{attribute 'linkalways'} 
{attribute 'no_explicit_call' := 'This FB is a CLASS and must be accessed using methods or properties'}
{attribute 'enable_dynamic_creation'}
FUNCTION_BLOCK PUBLIC DummyCommand EXTENDS AsyncCommand
VAR
	id : DINT;
	name : T_MaxString;
	timer : Ton;
END_VAR

METHOD PRIVATE AdsLog
VAR_INPUT
	message : T_MaxString;
END_VAR
VAR
	arrghhhh : T_MaxString := '%s';
END_VAR
VAR_INST
	format : FB_FormatString;
END_VAR
format(
	sFormat := 'DummyCommand{id=%d, name=%s} -> %s',
	arg1 := F_DInt(id),
	arg2 := F_String(name),
	arg3 := F_String(arrghhhh)
);

AdsLogStr(
	msgCtrlMask := ADSLOG_MSGTYPE_HINT,
	msgFmtStr := format.sOut,
	strArg := message
);
END_METHOD

METHOD FB_init : BOOL
VAR_INPUT
	bInitRetains : BOOL; // if TRUE, the retain variables are initialized (warm start / cold start)
	bInCopyCode : BOOL;  // if TRUE, the instance afterwards gets moved into the copy code (online change)
	id : DINT;
	name : T_MaxString;
END_VAR
THIS^.id := id;
THIS^.name := name;

AdsLog('FB_init');
END_METHOD

METHOD PROTECTED OnAborted
AdsLog('Aborted');
END_METHOD

METHOD PROTECTED OnAborting
VAR_INPUT
	stateControl : I_AsyncCommandStateControl;
END_VAR
AdsLog('Aborting');

WrapItUp(stateControl);
END_METHOD

METHOD PROTECTED OnCompleted : BOOL
AdsLog('Completed');
END_METHOD

METHOD PROTECTED OnCompleting
VAR_INPUT
	stateControl : I_AsyncCommandStateControl;
END_VAR
AdsLog('Completing');

WrapItUp(stateControl);
END_METHOD

METHOD PROTECTED OnErrored
VAR_INST
	firstCycle : BOOL;
END_VAR
IF NOT firstCycle THEN
	firstCycle := TRUE;
	AdsLog('Errored');
END_IF
END_METHOD

METHOD PROTECTED OnExecuting
VAR_INPUT
	stateControl : I_AsyncCommandStateControl;
END_VAR
VAR_INST
	firstCycle : BOOL;
END_VAR
IF NOT firstCycle THEN
	firstCycle := TRUE;
	AdsLog('Executing');
END_IF

timer(IN := TRUE, PT := T#10S);
IF timer.Q THEN
	stateControl.Next();
END_IF
END_METHOD

METHOD PROTECTED OnIdle
VAR_INST
	firstCycle : BOOL;
END_VAR
IF NOT firstCycle THEN
	firstCycle := TRUE;
	AdsLog('Idle');
END_IF
END_METHOD

METHOD PROTECTED OnInitializing
VAR_INPUT
	stateControl : I_AsyncCommandStateControl;
END_VAR
AdsLog('Initialising');

stateControl.Next();
END_METHOD

METHOD PUBLIC SimulateError
VAR_INPUT
	errorId : UDINT;
END_VAR
stateMachine.Error(errorId);
END_METHOD

METHOD PRIVATE WrapItUp
VAR_INPUT
	stateControl : I_AsyncCommandStateControl;
END_VAR
timer(IN := FALSE);
stateControl.Next();
END_METHOD

END_FUNCTION_BLOCK

(* stored: Version 1.1.0.1, ProductVersion 3.1.4024.12
   POU DummyCommand: Id {c45f4b59-19d8-459b-849f-afd6d76a0455}, SpecialFunc None
   Method AdsLog: Id {2ffffb3c-6af9-4aae-82d8-019d37b5655a}
   Method FB_init: Id {987e07d6-a661-461e-ad4f-6b7893904672}
   Method OnAborted: Id {044ca0ff-1d7a-474a-8927-4b64f87e9e38}
   Method OnAborting: Id {6d82c695-89af-42d6-9d3d-b8d4ebe09d5b}
   Method OnCompleted: Id {40545497-5659-48a8-b5ed-1031e09b5fca}
   Method OnCompleting: Id {b9ccf744-6791-4421-a4cc-cc862a85264e}
   Method OnErrored: Id {503aa4d3-2723-4bb3-b90a-fcecf0359d95}
   Method OnExecuting: Id {b004c861-4d1d-492e-a545-487079fe8580}
   Method OnIdle: Id {08430f16-a68e-4a5e-b45a-f35dc208c3f1}
   Method OnInitializing: Id {b77c0299-3327-4d59-b33b-2f995dc1885b}
   Method SimulateError: Id {03a41147-adf6-494f-a89f-acdde40dc6b7}
   Method WrapItUp: Id {d6b2a4de-4842-4e0b-82e3-b0ce35eafe27} *)
